{attribute 'qualified_only'}
VAR_GLOBAL CONSTANT
	ShortStringSize : UXINT := 80;
	LongStringSize : UXINT := 255;
END_VAR

(* stored: Version 1.1.0.1, ProductVersion 3.1.4024.4
   GVL Param_Configurations: Id {9f14be4b-a36a-4174-b8cc-72e6d57b2fba}, ParameterList True *)
